# EPICS substitutions: apps/amqApp/Db/amqDaq.substitutions
file "db/amqFloatArray.db" {
pattern    { P K N TH THH HSV HHSV }
    { B_DAQ:EB6:stats STA:EBDAQ6 4 10 20 MINOR MAJOR }
    { B_DAQ:EB2:stats STA:EBDAQ2 4 10 20 MINOR MAJOR }
}

file "db/array-to-scalar-4.template" {
pattern    { INP P FTVL }
    { B_DAQ:EB6:stats B_DAQ:EB6:stats: FLOAT }
    { B_DAQ:EB2:stats B_DAQ:EB2:stats: FLOAT }
}
